TYPE TcoDatamanStatus_v_5_x_x : STRUCT
    ActionDescription : STRING(100);
    ResultString : STRING;
    SignalStatus : TcoDatamanSignalStates_v_5_x_x;
END_STRUCT
END_TYPE

(* stored: Version 1.1.0.1, ProductVersion 3.1.4024.12
   DUT TcoDatamanStatus_v_5_x_x: Id {0627f38a-6166-047e-097c-aa383868e19b} *)
